FUNCTION_BLOCK ANY2ANY_2559F3670C2742D4 (* Any to any conversion *)
  (* Standard: 61499-2 *)
  (* Version 1.1, 24.06.2019, winkhub, nxtControl GmbH, support fixed STRING and UDT *)
  PACKAGE UAO.Hackathon;
  (* Compiler Cpp *)
  {SET_ATTRIBUTE(Runtime.FBType.ImplementingType, Runtime.Standard#DYNGEN_ANY2ANY)}
  {SET_ATTRIBUTE(Configuration.GenericFBType.InterfaceParams, Runtime.Standard#CNT:=1;IN${CNT$}:BOOL;OUT${CNT$}:USINT)}
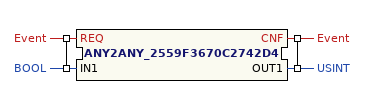
  EVENT_INPUT
    REQ WITH IN1; (* Normal Execution Request *)
  END_EVENT
  EVENT_OUTPUT
    CNF WITH OUT1; (* Execution Confirmation *)
  END_EVENT
  VAR_INPUT
    IN1 : BOOL; (* Argument *)
  END_VAR
  VAR_OUTPUT
    OUT1 : USINT; (* Result *)
  END_VAR
  EC_STATES
    START;
  END_STATES
END_FUNCTION_BLOCK
